// TIA Portal V20 export
TYPE "UserDiag_typeDiagnostics"
TITLE = UserDiag_typeDiagnostics
   STRUCT
      subfunctionStatus : Word := 16#0000;   // Block status or error information
      instructionError : Int := 0;   // Indicates in which system function the error occurred. 1:DeviceStates PN; 2=GetName PN; 3:ModuleStates PN; 4:DeviceStates DP; 5:GetName DP; 6:ModuleStates DP
      errorIndex : Int := 0;   // The last index of the respective loop, if an error occures (relevant for IOSystemCheck FB)
   END_STRUCT;
END_TYPE
